Staubli VAL3: goTo.pgx

program goTo(point x_pPoint, num x_nIndex, bool& x_bUnreached[], string x_sName, num x_nMoveType)
  local bool l_bUnreached
  local num l_nIndexTool
  local tool l_tTool
  local num l_nMoveType
  local mdesc l_mDesc
begin
  // look for not cycle mode
  if !cycleStatus:bCycle
    if cycleStatus:nWorkingMode==1 and isPowered()
      // check for the index
      if nOldIndex!=x_nIndex or (cycleStatus:nWorkingStatus!=0 and cycleStatus:nWorkingStatus!=6)
        if !isEmpty()
          resetMotion()
        endIf
        if nOldIndex!=x_nIndex
          nOldIndex=x_nIndex
        endIf
      else
        if isEmpty() and cycleStatus:nWorkingStatus==0
          // get the data to move
          call getTrajTool(l_tTool,sml:box[x_sName].nIndexGun)
          // use a sTemp mdesc to set the blend off
          l_mDesc.blend=off
          l_mDesc.accel=l_mDesc.decel=10
          l_mDesc.vel=10
          // use the got to of the trajectory...
          call MoveTo(x_pPoint,l_tTool,l_mDesc,x_nMoveType,x_bUnreached)
        endIf
      endIf
    else
      if cycleStatus:nWorkingMode!=1
        resetMotion()
      endIf
    endIf
  endIf
end
